// Mitsubishi GX Works2 project: HingeCutter   PLC: FX1N/FX1NC

TYPE Axis : STRUCT
  DirInstruction : BOOL;  (* bool Direction of pulse instruction *)
  Limited : BOOL;  (* bool Limit reached *)
  CurPos : DINT;  (* int Current position (mm) *)
  CurPosP : DINT;  (* int Current position (pulse) *)
  TarPos : DINT;  (* int Target position (mm) *)
  ManualN : BOOL;  (* bool Manual run: Negative direction *)
  ManualP : BOOL;  (* bool Manual run: Possitive direction *)
  ILimitN : BOOL;
  ILimitP : BOOL;
  OOnOff : BOOL;
  OReset : BOOL;
  OPulse : BOOL;
  ODirection : BOOL;
  TarR : BOOL;  (* bool Target reached *)
  Manual : BOOL;  (* bool Manual run: *)
  RunLatch : BOOL;
  RunLatchFalling : BOOL;
  Dir : BOOL;  (* bool Direction *)
  DirInt : DINT;  (* int Direction *)
  CurFS : DINT;  (* int Current feed speed *)
END_STRUCT END_TYPE

// global labels: Global1
VAR_GLOBAL
  CommandLtArray AT D100 : ARRAY [0..49] OF INT;
  TargetArrayX AT D200 : ARRAY [0..49] OF DINT;
  TargetArrayY AT D300 : ARRAY [0..49] OF DINT;
  FeedSpeedArrayX AT D400 : ARRAY [0..49] OF DINT;
  IsOn AT M0 : BOOL;
  RunButton AT M8 : BOOL;
  RunButtonRisingLatch : BOOL;
  RunButtonFallingLatch : BOOL;
  StopButton AT M9 : BOOL;
  ResetButton AT M2 : BOOL;
  SetButton AT M5 : BOOL;
  OriginButton AT M7 : BOOL;
  FeedSpeed AT D0 : DINT;
  OnOffResetStop : OnOffResetStop;
  XX : Axis;
  ManualHandler : ManualHandler;
  YY : Axis;
  OriginSetMove : OriginSetMove;
  FoilBlocker AT M14 : BOOL;
  PositionUpdater : PositionUpdater;
  AutoHandler : AutoHandler;
  PulseOutAndLimit : PulseOutAndLimit;
  AutoNextLine AT M10 : BOOL;
  FileEnded AT M11 : BOOL;
  ArrayIndex AT D10 : DINT;
  ArrayLength AT D16 : DINT;
  FeedSpeedArrayY AT D500 : ARRAY [0..49] OF DINT;
  CommandNbArray AT D150 : ARRAY [0..49] OF INT;
  CommandLt AT D17 : INT;
  CommandNb AT D18 : INT;
  ArrayIndexLimit AT D12 : DINT;
  ArrayIndexMax AT D14 : DINT;
  FoilClamper AT M15 : BOOL;
  Cutter1A AT M16 : BOOL;
  Cutter1B AT M17 : BOOL;
  Cutter2A AT M20 : BOOL;
  CommandHandler : CommandHandler;
  Cutter2B AT M21 : BOOL;
  Cutter3A AT M22 : BOOL;
  Cutter3B AT M23 : BOOL;
  OFoilBlocker AT Y004 : BOOL;
  OFoilClamper AT Y005 : BOOL;
  OCutter1A AT Y006 : BOOL;
  OCutter1B AT Y007 : BOOL;
  OCutter2A AT Y010 : BOOL;
  OCutter2B AT Y011 : BOOL;
  OCutter3A AT Y012 : BOOL;
  OCutter3B AT Y013 : BOOL;
END_VAR

// task Task_01 (event TRUE, interval 0, priority 31): POU_01

PROGRAM POU_01
OnOffResetStop();

IF IsOn THEN
	PositionUpdater();
	ManualHandler();
	AutoHandler();

	PulseOutAndLimit(fRunStart := RunButtonRisingLatch);
	
	RunButtonRisingLatch := FALSE;
	RunButtonFallingLatch := FALSE;
	RST(XX.TarR AND YY.TarR, RunButton);
	
	OriginSetMove();
END_IF;
END_PROGRAM

FUNCTION_BLOCK PulseOutAndLimit
VAR_INPUT
  fRunStart : BOOL;
END_VAR
(*X Axis ||||||||||||||||||||||||||||||||||||||||*)
OUT(XX.DirInt > 0, XX.Dir);
RST((NOT XX.ILimitN AND XX.Dir) OR (NOT XX.ILimitP AND NOT XX.Dir) OR (XX.ILimitN AND XX.ILimitP), XX.Limited);

DPLSV(XX.Manual AND NOT XX.Limited, FeedSpeed * XX.DirInt, XX.OPulse, XX.DirInstruction);

SET(fRunStart, XX.RunLatch);
DDRVA(XX.RunLatch AND NOT XX.Limited, XX.TarPos, XX.CurFS, XX.OPulse, XX.DirInstruction);
RST(M8029, XX.RunLatch);
PLF(XX.RunLatch, XX.RunLatchFalling);
SET(XX.RunLatchFalling, XX.TarR);
OUT(NOT XX.DirInstruction, XX.ODirection);

IF XX.RunLatch THEN
	XX.Dir := XX.DirInstruction;
END_IF;
SET((NOT XX.ILimitN AND NOT XX.Dir) OR (NOT XX.ILimitP AND XX.Dir), XX.Limited);
RST(XX.Limited, XX.RunLatch);

(*Y Axis ||||||||||||||||||||||||||||||||||||||||*)
OUT(YY.DirInt > 0, YY.Dir);
RST((NOT YY.ILimitN AND YY.Dir) OR (NOT YY.ILimitP AND NOT YY.Dir) OR (YY.ILimitN AND YY.ILimitP), YY.Limited);

DPLSV(YY.Manual AND NOT YY.Limited, FeedSpeed * YY.DirInt, YY.OPulse, YY.DirInstruction);

SET(fRunStart, YY.RunLatch);
DDRVA(YY.RunLatch AND NOT YY.Limited, YY.TarPos, YY.CurFS, YY.OPulse, YY.DirInstruction);
RST(M8029, YY.RunLatch);
PLF(YY.RunLatch, YY.RunLatchFalling);
SET(YY.RunLatchFalling, YY.TarR);
OUT(NOT YY.DirInstruction, YY.ODirection);

IF YY.RunLatch THEN
	YY.Dir := YY.DirInstruction;
END_IF;
SET((NOT YY.ILimitN AND NOT YY.Dir) OR (NOT YY.ILimitP AND YY.Dir), YY.Limited);
RST(YY.Limited, YY.RunLatch);
END_FUNCTION_BLOCK

FUNCTION_BLOCK OnOffResetStop
OUT(IsOn, XX.OOnOff);
OUT(IsOn, YY.OOnOff);

SET(ResetButton, XX.OReset);
SET(ResetButton, YY.OReset);
OUT_T(ResetButton, TC200, 8);
RST(TC200, ResetButton);
RST(TC200, XX.OReset);
RST(TC200, YY.OReset);

IF StopButton THEN
	RunButton := FALSE;
	XX.TarR := FALSE;
	XX.RunLatch := FALSE;
	YY.TarR := FALSE;
	YY.RunLatch := FALSE;
	FileEnded := FALSE;
	AutoNextLine := FALSE;
	StopButton := FALSE;
END_IF;
END_FUNCTION_BLOCK

FUNCTION_BLOCK OriginSetMove
VAR
  SetOrigin : BOOL;
  MoveToOrigin : BOOL;
END_VAR
OUT(OriginButton AND SetButton, SetOrigin);
OUT(OriginButton AND NOT SetButton, MoveToOrigin);

RST(SetOrigin, XX.CurPos);
RST(SetOrigin, XX.CurPosP);
RST(SetOrigin, YY.CurPos);
RST(SetOrigin, YY.CurPosP);
RST(SetOrigin, SetButton);

RST(MoveToOrigin, XX.TarPos);
RST(MoveToOrigin, YY.TarPos);
SET(MoveToOrigin, RunButton);

RST(SetOrigin OR MoveToOrigin, OriginButton);
END_FUNCTION_BLOCK

FUNCTION_BLOCK ManualHandler
IF NOT (RunButton OR AutoNextLine) THEN
	DMOV(XX.ManualN, -1, XX.DirInt);
	DMOV(XX.ManualP, 1, XX.DirInt);
	XX.Manual := XX.ManualN OR XX.ManualP;
	
	DMOV(YY.ManualN, -1, YY.DirInt);
	DMOV(YY.ManualP, 1, YY.DirInt);
	YY.Manual := YY.ManualN OR YY.ManualP;
END_IF;
RST(RunButton, XX.Manual);
RST(RunButton, YY.Manual);
END_FUNCTION_BLOCK

FUNCTION_BLOCK AutoHandler
VAR
  fRunButtonFalling : BOOL;
  fRunButtonRising : BOOL;
END_VAR
PLS(RunButton, fRunButtonRising);
SET(fRunButtonRising, RunButtonRisingLatch);
PLF(RunButton, fRunButtonFalling);
SET(fRunButtonFalling, RunButtonFallingLatch);

IF RunButtonRisingLatch THEN
	CommandHandler();
	
	DMOV(NOT AutoNextLine, FeedSpeed, XX.CurFS);
	DMOV(NOT AutoNextLine, FeedSpeed, YY.CurFS);
	
	XX.TarR := XX.CurPos = XX.TarPos;
	YY.TarR := YY.CurPos = YY.TarPos;

	RST(XX.TarR AND YY.TarR, RunButton);
END_IF;

IF RunButtonFallingLatch AND AutoNextLine THEN
	SET(ArrayIndex > ArrayIndexLimit, FileEnded);
	IF (ArrayIndex < ArrayIndexLimit) OR (ArrayIndex = ArrayIndexMax) THEN
		CommandLt := CommandLtArray[ArrayIndex];
		CommandNb := CommandNbArray[ArrayIndex];
		XX.TarPos := TargetArrayX[ArrayIndex];
		YY.TarPos := TargetArrayY[ArrayIndex];
		XX.CurFS := FeedSpeedArrayX[ArrayIndex];
		YY.CurFS := FeedSpeedArrayY[ArrayIndex];
		ArrayIndex := ArrayIndex + 1;
	END_IF;
	XX.TarR := FALSE;
	YY.TarR := FALSE;
	RunButton := NOT FileEnded;
	RST(FileEnded, AutoNextLine);
END_IF;
END_FUNCTION_BLOCK

FUNCTION_BLOCK PositionUpdater
XX.CurPos := XX.CurPosP;
YY.CurPos := YY.CurPosP;
END_FUNCTION_BLOCK

FUNCTION_BLOCK CommandHandler
(**)
RST(CommandLt = 0 AND CommandNb = 0, FoilBlocker);
SET(CommandLt = 0 AND CommandNb = 1, FoilBlocker);
OUT(FoilBlocker, OFoilBlocker);
(**)
RST(CommandLt = 1 AND CommandNb = 0, FoilClamper);
SET(CommandLt = 1 AND CommandNb = 1, FoilClamper);
OUT(FoilClamper, OFoilClamper);
(**)
RST(CommandLt = 2 AND CommandNb = 0, Cutter1A);
RST(CommandLt = 2 AND CommandNb = 0, Cutter1B);
SET(CommandLt = 2 AND CommandNb = 1, Cutter1A);
RST(CommandLt = 2 AND CommandNb = 1, Cutter1B);
SET(CommandLt = 2 AND CommandNb = 2, Cutter1A);
SET(CommandLt = 2 AND CommandNb = 2, Cutter1B);
OUT(Cutter1A, OCutter1A);
OUT(Cutter1B, OCutter1B);
(**)
RST(CommandLt = 3 AND CommandNb = 0, Cutter2A);
RST(CommandLt = 3 AND CommandNb = 0, Cutter2B);
SET(CommandLt = 3 AND CommandNb = 1, Cutter2A);
RST(CommandLt = 3 AND CommandNb = 1, Cutter2B);
SET(CommandLt = 3 AND CommandNb = 2, Cutter2A);
SET(CommandLt = 3 AND CommandNb = 2, Cutter2B);
OUT(Cutter2A, OCutter2A);
OUT(Cutter2B, OCutter2B);
(**)
RST(CommandLt = 4 AND CommandNb = 0, Cutter3A);
RST(CommandLt = 4 AND CommandNb = 0, Cutter3B);
SET(CommandLt = 4 AND CommandNb = 1, Cutter3A);
RST(CommandLt = 4 AND CommandNb = 1, Cutter3B);
SET(CommandLt = 4 AND CommandNb = 2, Cutter3A);
SET(CommandLt = 4 AND CommandNb = 2, Cutter3B);
OUT(Cutter3A, OCutter3A);
OUT(Cutter3B, OCutter3B);
END_FUNCTION_BLOCK
